// TIA Portal V20 export
TYPE "AnalogInput_DT"
   STRUCT
      SWRealValue : Real;   // Software real value use in PLC
      HWWordValue : Word;   // Hardware value direclty from physical input
   END_STRUCT;
END_TYPE
